// TIA Portal V20 export
FUNCTION_BLOCK "DataTakeOver"   // FB302, FBD
{ S7_Optimized_Access := 'TRUE' }
// stored: AutoNumber false, MemoryReserve 100, SetENOAutomatically false
   VAR
      Var { ExternalAccessible := 'False'; ExternalVisible := 'False'; ExternalWritable := 'False'} : "TypeVar";
   END_VAR
BEGIN

REGION Network 1 (SCL): config data from pc
   IF "ComRd".Data.Config.active AND "G".comOk THEN

       // config for mode
       "G".Cfg.adjScannerActive := "ComRd".Data.Config.adjScannerActive;
       "G".Cfg.adjTopActive := "ComRd".Data.Config.adjTopActive;
       "G".Cfg.adjLeftActive := "ComRd".Data.Config.adjLeftActive;
       "G".Cfg.adjRightActive := "ComRd".Data.Config.adjRightActive;

       "G".Cfg.adjTopActiveLinMot := "ComRd".Data.Config.adjTopLinMotActive;
       "G".Cfg.adjLeftActiveLinMot := "ComRd".Data.Config.adjLeftLinMotActive;
       "G".Cfg.adjRightActiveLinMot := "ComRd".Data.Config.adjRightLinMotActive;

       "G".Cfg.xrayActive := "ComRd".Data.Config.xrayActive ;

       // config for mode
       "G".Cfg.modeBoardPassing:= "ComRd".Data.Config.modeBoardPassing;
       "G".Cfg.modeDimension := "ComRd".Data.Config.modeDimension;
       "G".Cfg.modeRandomAdj := "ComRd".Data.Config.modeRandomAdj;

       // config for sensor for random adjustment
       IF "ComRd".Data.Config.modeDimension = 3 OR "ComRd".Data.Config.modeDimension = 4 THEN
           "G".Cfg.senTopActive := TRUE;
       ELSE
           "G".Cfg.senTopActive := FALSE;
       END_IF;
       IF "ComRd".Data.Config.modeDimension = 2 OR "ComRd".Data.Config.modeDimension = 4 THEN
           IF "ComRd".Data.Config.modeBoardPassing = 3 THEN
               "G".Cfg.senLeftActive := TRUE;
               "G".Cfg.senRightActive := TRUE;
           ELSIF "ComRd".Data.Config.modeBoardPassing = 2 THEN
               "G".Cfg.senLeftActive := TRUE;
               "G".Cfg.senRightActive := FALSE;
           ELSIF "ComRd".Data.Config.modeBoardPassing = 1 THEN
               "G".Cfg.senLeftActive := FALSE;
               "G".Cfg.senRightActive := TRUE;
           END_IF;
       ELSE
           "G".Cfg.senLeftActive := FALSE;
           "G".Cfg.senRightActive := FALSE;
       END_IF;

       // config for encoder 1
       IF "ComRd".Data.Config.enc1QuadEvalActive THEN
           "G".Cfg.enc1Gain := (1.0 / INT_TO_REAL("ComRd".Data.Config.enc1Factor)) * 1.0;
       ELSE
           "G".Cfg.enc1Gain := (1.0 / INT_TO_REAL("ComRd".Data.Config.enc1Factor)) * 1.0;
       END_IF;
       IF "ComRd".Data.Config.enc1Factor = -1 THEN
           "G".Cfg.enc1Active := FALSE;
       ELSE
           "G".Cfg.enc1Active := TRUE;
       END_IF;

   END_IF;
END_REGION

REGION Network 2 (SCL): batch from pc
   IF "G".comOk THEN
       // Width
       IF "ComRd".Data.batch.MinWidth = "ComRd".Data.batch.MaxWidth THEN
           "G".Batch.widthMin := DINT_TO_REAL("ComRd".Data.batch.MinWidth) / 10.0;
           "G".Batch.widthMax := DINT_TO_REAL("ComRd".Data.batch.MaxWidth) / 10.0;
           "G".Batch.width := DINT_TO_REAL("ComRd".Data.batch.MinWidth) / 10.0;
       ELSIF "ComRd".Data.batch.MinWidth <> "ComRd".Data.batch.MaxWidth THEN
           "G".Batch.widthMin := DINT_TO_REAL("ComRd".Data.batch.MinWidth) / 10.0;
           "G".Batch.widthMax := DINT_TO_REAL("ComRd".Data.batch.MaxWidth) / 10.0;
           "G".Batch.width := DINT_TO_REAL(("ComRd".Data.batch.MinWidth + "ComRd".Data.batch.MaxWidth) / 2) / 10.0;
       END_IF;

       // Thickness
       IF "ComRd".Data.batch.MinThickness = "ComRd".Data.batch.MaxThickness THEN
           "G".Batch.thicknessMin := DINT_TO_REAL("ComRd".Data.batch.MinThickness) / 10.0;
           "G".Batch.thicknessMax := DINT_TO_REAL("ComRd".Data.batch.MaxThickness) / 10.0;
           "G".Batch.thickness := DINT_TO_REAL("ComRd".Data.batch.MinThickness) / 10.0;
       ELSIF "ComRd".Data.batch.MinThickness <> "ComRd".Data.batch.MaxThickness THEN
           "G".Batch.thicknessMin := DINT_TO_REAL("ComRd".Data.batch.MinThickness) / 10.0;
           "G".Batch.thicknessMax := DINT_TO_REAL("ComRd".Data.batch.MaxThickness) / 10.0;
           "G".Batch.thickness := DINT_TO_REAL(("ComRd".Data.batch.MinThickness + "ComRd".Data.batch.MaxThickness) / 2) / 10.0;
       END_IF;
   END_IF;
END_REGION
END_FUNCTION_BLOCK
